(* CODESYS project Estação 7 - Storage (2022).project

Project tree, tasks and I/O mapping:
  Device : CPX-CEC-C1-V3, Festo AG & Co. KG, order no. 3473128, version 3.5.7.37
      unmapped channels: Rotary switch
    application Application
      libraries: Standard, * (System)
      task MainTask (cyclic, interval t#20ms, priority 20) calls PLC_PRG
      program PLC_PRG [ST]
      global variables GVL
      visualisation Visualization_1
      program entrada_pecas [ST]
      program pisca_pisca [ST]
      program home [ST]
      program processo [ST]
      program saida_pecas [ST]
      program atualizar_valores [ST]
      program teste_comunicacao [ST]
    PLC_Diagnosis : PLC-Diagnosis, Festo AG & Co. KG, version 3.5.4.1
    CPX_System : CPX_System, Festo AG & Co. KG, order no. 3473128, version 1.258
      CEC_C1_V3 : CEC-C1-V3, Festo AG & Co. KG, order no. 3473128, version 1.258
          settings:  = 0;  = 232080133852672;  = 1174579392;  = 65535;  = 16885952;  = 13959208;  = 1f5d13d3;  = 5
      _8DI_8DO : 8DI/8DO, Festo AG & Co. KG, order no. 526257, version 1.258
          settings:  = 0;  = 1;  = 1;  = 1;  = 1;  = 0;  = 1;  = 1;  = 0;  = 0;  = 0;  = 0;  = 0;  = 0;  = 0;  = 0;  = 0;  = 0;  = 0;  = 0;  = 0;  = 0;  = 0;  = 0;  = 0;  = 0;  = 0;  = 0;  = 0;  = 0;  = 0;  = 0;  = 0;  = 0;  = 0;  = 0;  = 0;  = 0;  = 0;  = 0;
             = 0;  = 0;  = 0;  = 0;  = 0;  = 0;  = 0;  = 0;  = 0;  = 0;  = 0;  = 0;  = 0;  = 0;  = 0;  = 0;  = 0;  = 0;  = 0;  = 0;  = 0;  = 0;  = 0;  = 0;  = 0;  = 0;  = 0;  = 0;  = 0;  = 0;  = 0;  = 0;  = 0;  = 0;  = 0;  = 0;  = 0;  = 0;  = 0;  = 0;
             = 576751027668385792;  = 'PI%i.0.0.1=1';  = 'PI%i.0.1.1=1';  = 'PI%i.0.2.1=1';  = 'PI%i.1.0.1=1';  = 'PI%i.1.1.1=0';  = 'PI%i.1.4.2=1';  = 'PI%i.1.6.2=1';  = 'PI%i.6.0.1=0';  = 'PI%i.6.1.1=0';  = 'PI%i.6.2.1=0';  = 'PI%i.6.3.1=0';  = 'PI%i.6.4.1=0';  = 'PI%i.6.5.1=0';  = 'PI%i.6.6.1=0';  = 'PI%i.6.7.1=0';  = dd30774a;  = 6
          unmapped channels: Input 0, Output 0
      _8DI_8DO_1 : 8DI/8DO, Festo AG & Co. KG, order no. 526257, version 1.258
          settings:  = 0;  = 1;  = 1;  = 1;  = 1;  = 0;  = 1;  = 1;  = 0;  = 0;  = 0;  = 0;  = 0;  = 0;  = 0;  = 0;  = 0;  = 0;  = 0;  = 0;  = 0;  = 0;  = 0;  = 0;  = 0;  = 0;  = 0;  = 0;  = 0;  = 0;  = 0;  = 0;  = 0;  = 0;  = 0;  = 0;  = 0;  = 0;  = 0;  = 0;
             = 0;  = 0;  = 0;  = 0;  = 0;  = 0;  = 0;  = 0;  = 0;  = 0;  = 0;  = 0;  = 0;  = 0;  = 0;  = 0;  = 0;  = 0;  = 0;  = 0;  = 0;  = 0;  = 0;  = 0;  = 0;  = 0;  = 0;  = 0;  = 0;  = 0;  = 0;  = 0;  = 0;  = 0;  = 0;  = 0;  = 0;  = 0;  = 0;  = 0;
             = 576751027668385792;  = 'PI%i.0.0.1=1';  = 'PI%i.0.1.1=1';  = 'PI%i.0.2.1=1';  = 'PI%i.1.0.1=1';  = 'PI%i.1.1.1=0';  = 'PI%i.1.4.2=1';  = 'PI%i.1.6.2=1';  = 'PI%i.6.0.1=0';  = 'PI%i.6.1.1=0';  = 'PI%i.6.2.1=0';  = 'PI%i.6.3.1=0';  = 'PI%i.6.4.1=0';  = 'PI%i.6.5.1=0';  = 'PI%i.6.6.1=0';  = 'PI%i.6.7.1=0';  = dd39f1d3;  = 6
          unmapped channels: Input 0, Output 0
    Ethernet : Ethernet, 3S - Smart Software Solutions GmbH, version 3.5.10.0
      ModbusTCP_Slave_Device : ModbusTCP Slave Device, 3S - Smart Software Solutions GmbH, version 3.5.10.0
          unmapped channels: Inputs, Outputs
  visualisation Visualization
  text list GlobalTextList
*)

// Device/Application/GVL
{attribute 'qualified_only'}
VAR_GLOBAL
//Entradas
//Sensores
	E_home 	AT %IX1.0 :BOOL; //
	E_error 	 	AT %IX1.1 :BOOL; //
	E_processo	AT %IX1.2 :BOOL; //
	Armazenagem_completada			AT %IX1.3 :BOOL;
	E_provesso 		AT %IX1.4  :BOOL; //
	S_cor 			AT %IX1.5  :BOOL; //Sensor para verificar se a peça é preta
	S_indutivo  	AT %IX1.6  :BOOL; //Sensor indutivo
	//S_indutivodadw 	AT %IX1.7  :BOOL; //Sensor indutivo
//IHM
	Start_btn 		AT	%IX2.0	:BOOL;  //Botão de start
	Stop_btn 		AT	%IX2.1	:BOOL;	//Botão de stop (NF)
	Chave 			AT	%IX2.2	:BOOL;	//Chave auto/manual
	Reset_btn 		AT	%IX2.3	:BOOL;	//Botão de reset
	I4_IHM			AT	%IX2.4	:BOOL;	//Bit de saída 4 da IHM
	I5_IHM			AT	%IX2.5	:BOOL;	//Bit de saída 5 da IHM
	S_Entrada 			AT	%IX2.6	:BOOL;	//Bit de saída 6 da IHM
	I7_IHM			AT	%IX2.7	:BOOL;	//Bit de saída 7 da IHM

	
//Saídas

	//Sinais para o CECC 			
	Fazer_home 	AT	%QX0.0	:BOOL;	//
	Reset_erro 	AT	%QX0.1	:BOOL;	//
	Modo_E_S 	AT	%QX0.2	:BOOL;	//
	B1		 	AT	%QX0.3	:BOOL;	
	B2 			AT	%QX0.4	:BOOL;	//
	B3		 	AT	%QX0.5	:BOOL;	
	gatilho		AT	%QX0.6	:BOOL;	
	Configuracao AT	%QX0.7	:BOOL;	

//IHM				
	Start_LED		AT	%QX1.0	:BOOL;	//LED do botão de start
	Reset_LED 		AT	%QX1.1	:BOOL;	//LED do botão de reset
	Q1_LED 			AT	%QX1.2	:BOOL;	//LED sinalizador Q1
	Q2_LED			AT	%QX1.3	:BOOL;	//LED sinalizador Q2
	E_Saindo		AT	%QX1.5	:BOOL;	//Saída Q4 IHM //Esteira entrando
	E_Entrando		AT	%QX1.4	:BOOL;	//Saída Q5 IHM //Esteira saindo
	Q6_IHM			AT	%QX1.6	:BOOL;	//Saída Q6 IHM
	Q7_IHM 			AT	%QX1.7	:BOOL;	//Saída Q7 IHM
	
	
	flag_btn_visu :BOOL;
	btn_armazena :  BOOL;
	
	B1_Modbus : BOOL;
	B2_Modbus : BOOL;
	B3_Modbus : BOOL;
	
	home: BOOL := FALSE; //Trigger para que a estação reset os erros e faça home
	ligar_pisca: BOOL := FALSE; //Flag para ligar e desligar o pisca pisca
	iniciar_processo: BOOL := FALSE; //Inicia a função de processo, onde pega ou retira a peça de acordo com a flag definir_sentido. Se essa flag estiver setada, é saída. 
	retirar_peca: BOOL := FALSE; //Flag para iniciar processo de retirada da peça (ligar a esteira para retirar a peça da estação 7 e jogar para a 6).
	definir_sentido:	BOOL := FALSE; //Flag para definir se a peça vai entrar ou saír.
	flag_primeira_entrada : BOOL := FALSE; //Flag para ajudar a gerenciar o sinal da saída Q7 da IHM
	estacao_iniciada : BOOL; //Falg para sinalizar que a estação está iniciada 
	estacao_parada: BOOL; //Flag para sinalizar que a estação está parada
	//MODBUS bits
	//Entradas
	Mod_I_0_0 		AT %IX4.0 : BOOL;//start 
	Mod_I_0_1	 	AT %IX4.1 : BOOL;//stop
	Mod_I_0_2 		AT %IX4.2 : BOOL;//reset
	Mod_I_0_3 		AT %IX4.3 : BOOL;//Modo entrada 
	Mod_I_0_4 		AT %IX4.4 : BOOL;//Modo saída 
	Mod_I_0_5 		AT %IX4.5 : BOOL;//Teste resposta da estação - IN 
	Mod_I_0_6 		AT %IX4.6 : BOOL;//B1
	Mod_I_0_7 		AT %IX4.7 : BOOL;//B2		

	Mod_I_1_0 		AT %IX5.0 : BOOL;//B3
	Mod_I_1_1	 	AT %IX5.1 : BOOL;//Iniciar processo
	Mod_I_1_2 		AT %IX5.2 : BOOL;//Confirmação de leitura das cores pela central
	Mod_I_1_3 		AT %IX5.3 : BOOL;
	Mod_I_1_4 		AT %IX5.4 : BOOL;
	Mod_I_1_5 		AT %IX5.5 : BOOL;
	Mod_I_1_6 		AT %IX5.6 : BOOL;
	Mod_I_1_7 		AT %IX5.7 : BOOL;
	
	//Saídas
	Mod_Q_0_0 		AT %QX2.0 : BOOL;//Estação iniciada 	
	Mod_Q_0_1	 	AT %QX2.1 : BOOL;// Estação parada 
	Mod_Q_0_2 		AT %QX2.2 : BOOL;//Estação em processo
	Mod_Q_0_3 		AT %QX2.3 : BOOL;// Estação em modo entrada 
	Mod_Q_0_4 		AT %QX2.4 : BOOL;// Estação em modo saída 
	Mod_Q_0_5 		AT %QX2.5 : BOOL;// Teste resposta da estação - OUT
	Mod_Q_0_6 		AT %QX2.6 : BOOL;//B1 - bit 0 da cor
	Mod_Q_0_7 		AT %QX2.7 : BOOL;//B2 - bit 1 da cor
	
	Mod_Q_1_0 		AT %QX3.0 : BOOL;//B3 - bit 2 da cor
	Mod_Q_1_1 		AT %QX3.1 : BOOL;//Sensor de entrada da estação
	Mod_Q_1_2 		AT %QX3.2 : BOOL;//Cor disponível para leitura
	Mod_Q_1_3 		AT %QX3.3 : BOOL; 
	Mod_Q_1_4 		AT %QX3.4 : BOOL; 
	Mod_Q_1_5	 	AT %QX3.5 : BOOL; 
	Mod_Q_1_6 		AT %QX3.6 : BOOL; 
	Mod_Q_1_7 		AT %QX3.7 : BOOL; 
	
	Mod_Q_2_0 		AT %QX4.0 : BOOL;
	Mod_Q_2_1 		AT %QX4.1 : BOOL;
	Mod_Q_2_2 		AT %QX4.2 : BOOL;
	Mod_Q_2_3 		AT %QX4.3 : BOOL; 
	Mod_Q_2_4 		AT %QX4.4 : BOOL;
	Mod_Q_2_5	 	AT %QX4.5 : BOOL;
	Mod_Q_2_6 		AT %QX4.6 : BOOL; 
	Mod_Q_2_7 		AT %QX4.7 : BOOL; 
	
	Mod_Q_3_0 		AT %QX5.0 : BOOL; //Teste de comunicação - resposta - BIT 24
	Mod_Q_3_1 		AT %QX5.1 : BOOL; 
	Mod_Q_3_2 		AT %QX5.2 : BOOL;
	Mod_Q_3_3 		AT %QX5.3 : BOOL; 
	Mod_Q_3_4 		AT %QX5.4 : BOOL; 
	Mod_Q_3_5	 	AT %QX5.5 : BOOL; 
	Mod_Q_3_6 		AT %QX5.6 : BOOL; 
	Mod_Q_3_7 		AT %QX5.7 : BOOL;
	
END_VAR

// Device/Application/PLC_PRG
PROGRAM PLC_PRG
VAR

	
	
	
END_VAR

atualizar_valores(); //Função que atualiza as variáveis e o MODBUS
pisca_pisca(); //Função que permite o pisca pisca rodar
home(); //Função para fazer o HOME da estação
teste_comunicacao(); //Função para teste de comunicação

IF NOT gvl.estacao_parada AND gvl.estacao_iniciada THEN //Caso a estação não esteja parada e esteja iniciada
	entrada_pecas(); //Função de entrada de peças
	processo(); 	 //Função de processo 
	saida_pecas();   //Função de saída de peças
	gvl.Q1_LED := TRUE; //Liga o LED que indica estação iniciada
ELSE
	gvl.E_Entrando := FALSE; //Reseta flag que indica peça entrando
	gvl.E_Saindo := FALSE;	//Reseta a flag que indica peça saindo	
	gvl.ligar_pisca := FALSE; //Reseta flag que inicia o pisca pisca
	gvl.Q1_LED := FALSE;	 //Apaga o LED que inidca que a estação está iniciada
END_IF

gvl.Modo_E_S := gvl.definir_sentido; //Define entrada ou saída

END_PROGRAM

// Device/Application/atualizar_valores
PROGRAM atualizar_valores
VAR
END_VAR

GVL.Mod_Q_0_0 := GVL.estacao_iniciada; 
GVL.Mod_Q_0_1 := GVL.estacao_parada;
//GVL.Mod_Q_0_2 := GVL.E_processo;
gvl.Mod_Q_0_2 := gvl.ligar_pisca;

IF GVL.definir_sentido THEN
	GVL.Mod_Q_0_3 := FALSE;
	GVL.Mod_Q_0_4 := TRUE;
	ELSE
	GVL.Mod_Q_0_3 := TRUE;
	GVL.Mod_Q_0_4 := FALSE;
END_IF


GVL.Mod_Q_0_6 := GVL.B1_Modbus;
GVL.Mod_Q_0_7 := GVL.B2_Modbus;
GVL.Mod_Q_1_0 := GVL.B3_Modbus;


gvl.iniciar_processo := gvl.Mod_I_1_1; //ATUALIZADO

IF GVL.Mod_I_0_3 AND NOT gvl.Mod_I_0_4 THEN //Sentido de entrada de peças //ATUALIZADO
	gvl.definir_sentido := FALSE;
END_IF

IF NOT GVL.Mod_I_0_3 AND  gvl.Mod_I_0_4 THEN //Sentido de saída de peças //ATUALIZADO
	gvl.definir_sentido := TRUE;
	gvl.B1 := GVL.Mod_I_0_6;//ATUALIZADO
	gvl.B2 := GVL.Mod_I_0_7;//ATUALIZADO
	gvl.B3 := GVL.Mod_I_1_0;//ATUALIZADO
END_IF

IF GVL.Reset_btn OR GVL.Mod_I_0_2 THEN  //Reset geral e home da estação //ATUALIZADO
	gvl.home  := TRUE;
	GVL.estacao_parada := false;
END_IF

IF NOT GVL.Stop_btn OR GVL.Mod_I_0_1 THEN 
	GVL.estacao_parada := TRUE;
END_IF

IF GVL.Start_btn OR GVL.Mod_I_0_0 THEN 
	if not gvl.estacao_parada then
		gvl.estacao_iniciada := true;
	END_IF
END_IF

IF gvl.Mod_I_1_2 THEN
	GVL.B1_Modbus := FALSE;
	GVL.B2_Modbus := FALSE;
	GVL.B3_Modbus := FALSE;
	GVL.Mod_Q_1_2 := FALSE;
END_IF

END_PROGRAM

// Device/Application/home
PROGRAM home
VAR
	
	TON_temp_1: TON;
	TON_1: BOOL;
	TON_temp_2: TON;
	TON_2: BOOL;
	
	passo: INT;

END_VAR

TON_temp_1(IN := TON_1, PT:= T#0.4S);
TON_temp_2(IN := TON_2, PT:= T#0.4S);

IF  gvl.home THEN  //Reset geral da estação
	gvl.ligar_pisca := TRUE;
	GVL.Reset_erro := TRUE;	
	TON_1 := TRUE;
	passo := 1;
	gvl.home := FALSE;
	GVL.Fazer_home := TRUE;	
END_IF

IF TON_temp_1.Q  AND (passo = 1) THEN //Home
	passo := 0;
	GVL.Reset_erro := FALSE;
	GVL.Fazer_home := TRUE;	
	TON_1 := FALSE;
	TON_2 := TRUE;
	passo := 2;
END_IF

IF TON_temp_2.Q  AND  (passo = 2) THEN //Finalização da home
	GVL.Fazer_home := FALSE;	
	TON_2 := FALSE;
	passo := 3;
END_IF

IF (passo = 3) AND NOT gvl.E_processo THEN
	passo := 0;
	gvl.ligar_pisca := FALSE;
END_IF

END_PROGRAM

// Device/Application/pisca_pisca
PROGRAM pisca_pisca
VAR
	
	TON_temp_1: TON;
	TON_1: BOOL;
	TON_temp_2: TON;
	TON_2: BOOL;
	
	passo: INT;
END_VAR

TON_temp_1(IN := TON_1, PT:= T#0.2S);
TON_temp_2(IN := TON_2, PT:= T#0.2S);

IF gvl.ligar_pisca AND (passo = 0)  THEN
	TON_1 := TRUE;
	passo := 1;
END_IF

IF NOT gvl.ligar_pisca THEN
	TON_1 := FALSE;
	TON_2 := FALSE;
	GVL.Q2_LED := FALSE;
	passo := 0;
END_IF

IF TON_temp_1.Q THEN
	TON_1 := FALSE;
	TON_2 := TRUE;
	GVL.Q2_LED := TRUE;
END_IF

IF TON_temp_2.Q THEN
	TON_1 := TRUE;
	TON_2 := FALSE;
	GVL.Q2_LED := FALSE;
END_IF

END_PROGRAM

// Device/Application/teste_comunicacao
PROGRAM teste_comunicacao
VAR
	
	TON_temp_1: TON;
	TON_1: BOOL;	

END_VAR

gvl.Mod_Q_0_5 := gvl.Mod_I_0_5;

END_PROGRAM

// Device/Application/entrada_pecas
PROGRAM entrada_pecas
VAR
	PASSOS_LETURA: INT;
	
	TON_temp_1: TON;
	TON_1: BOOL;
	
	TON_temp_2: TON;
	TON_2: BOOL;
	
	TON_temp_esteira: TON;
	TON_esteira: BOOL;
	
	METALICO: BOOL;
	REFLETE: BOOL;
	
	
END_VAR

TON_temp_1(IN := TON_1, PT:= T#0.4S);
TON_temp_2(IN := TON_2, PT:= T#0.4S);
//Timer para a chagada da peça no sensor da esteira (Esse sensor não está ligado ao CPX, então não consigo utilizar o sinal dele)
TON_temp_esteira(IN := TON_esteira, PT:= T#3S);

IF NOT gvl.definir_sentido AND NOT gvl.E_processo AND NOT gvl.flag_primeira_entrada THEN
	gvl.Q7_IHM := TRUE; 
	gvl.flag_primeira_entrada := TRUE;
END_IF

IF gvl.S_Entrada AND (PASSOS_LETURA = 0) AND NOT gvl.definir_sentido THEN
	gvl.ligar_pisca := TRUE;
	gvl.E_Entrando := TRUE;
	PASSOS_LETURA := 1;
	TON_esteira := TRUE;
	gvl.Q7_IHM := FALSE; 
END_IF

IF (PASSOS_LETURA = 1) AND NOT TON_temp_esteira.Q THEN
	IF NOT METALICO THEN
		METALICO := gvl.S_indutivo;
	END_IF
	IF NOT REFLETE THEN
		REFLETE := gvl.S_cor;
	END_IF
	
END_IF

IF (PASSOS_LETURA = 1) AND  TON_temp_esteira.Q THEN
	
	GVL.B1_Modbus := FALSE;
	GVL.B2_Modbus := FALSE;
	GVL.B3_Modbus := FALSE;
	GVL.Mod_Q_1_2 := FALSE;

	PASSOS_LETURA := 0;
	TON_esteira := FALSE;
	gvl.E_Entrando := FALSE;
	IF METALICO THEN 	
		GVL.B1	:= FALSE;
		GVL.B2	:= TRUE;
		GVL.B3  := FALSE;
	END_IF
	IF NOT METALICO AND REFLETE THEN 	
		GVL.B1	:= FALSE;
		GVL.B2	:= FALSE;
		GVL.B3  := FALSE;
	END_IF
	IF NOT METALICO AND NOT REFLETE THEN 	
		GVL.B1	:= TRUE;
		GVL.B2	:= FALSE;
		GVL.B3  := FALSE;
	END_IF
	
	GVL.B1_Modbus := GVL.B1;
	GVL.B2_Modbus := GVL.B2;
	GVL.B3_Modbus := GVL.B3;
	GVL.Mod_Q_1_2 := TRUE;
	
	METALICO := FALSE;
	REFLETE := FALSE;
	
	PASSOS_LETURA := 2;
END_IF

IF (PASSOS_LETURA = 2) AND NOT gvl.E_processo THEN
	PASSOS_LETURA := 0;
	gvl.iniciar_processo := TRUE;
END_IF

END_PROGRAM

// Device/Application/processo
PROGRAM processo
VAR
	
vetor: INT;
	
	TON_temp_1: TON;
	TON_1: BOOL;
	
	TON_temp_2: TON;
	TON_2: BOOL;
	
	PASSOS: INT;

END_VAR

TON_temp_1(IN := TON_1, PT:= T#0.4S);
TON_temp_2(IN := TON_2, PT:= T#0.4S);

IF NOT gvl.E_processo   AND (GVL.btn_armazena  OR (gvl.iniciar_processo)) THEN
	gvl.iniciar_processo := FALSE;
	gvl.ligar_pisca := TRUE;
	gvl.Configuracao := TRUE;
	TON_1 := TRUE;
	PASSOS := 1;
	
END_IF

IF (PASSOS = 1) AND TON_temp_1.Q THEN
	PASSOS := 2;
	TON_1 := FALSE;
	TON_2 := TRUE;
END_IF

IF (PASSOS = 2) AND TON_temp_2.Q THEN
	PASSOS := 3;
	TON_2 := FALSE;
	gvl.gatilho := TRUE;	
	TON_1 := TRUE;
END_IF

IF (PASSOS = 3) AND TON_temp_1.Q THEN
	PASSOS := 4;
	TON_1 := FALSE;
	gvl.gatilho := FALSE;
	TON_2 := TRUE;
END_IF

IF (PASSOS = 4) AND TON_temp_2.Q THEN
	PASSOS := 5;
	TON_2 := FALSE;
	GVL.B1	:= FALSE;
	GVL.B2	:= FALSE;
	GVL.B3  := FALSE;
END_IF

IF (PASSOS = 5) AND NOT gvl.E_processo THEN
	PASSOS := 0;
	gvl.iniciar_processo := FALSE;
	gvl.ligar_pisca := FALSE;
	gvl.flag_primeira_entrada := FALSE;
	IF gvl.Modo_E_S THEN
		gvl.retirar_peca := TRUE;
	END_IF 
	IF NOT gvl.Modo_E_S THEN
		gvl.Q7_IHM := TRUE;
	END_IF
END_IF

END_PROGRAM

// Device/Application/saida_pecas
PROGRAM saida_pecas
VAR

	PASSOS: INT;
	
	TON_temp_esteira: TON;
	TON_esteira: BOOL;
	
	TON_temp_1: TON;
	TON_1: BOOL;	
	
	METALICO: BOOL;
	REFLETE: BOOL;	

END_VAR

TON_temp_1(IN := TON_1, PT:= T#0.8S);
//Timer para a chagada da peça no sensor da esteira (Esse sensor não está ligado ao CPX, então não consigo utilizar o sinal dele)
TON_temp_esteira(IN := TON_esteira, PT:= T#3S);

IF gvl.retirar_peca AND (PASSOS = 0)THEN
	gvl.retirar_peca := FALSE;
	gvl.ligar_pisca := TRUE;
	gvl.E_saindo := TRUE;
	gvl.Q7_IHM := FALSE;
	PASSOS := 1;
END_IF

IF (PASSOS = 1) AND gvl.S_Entrada THEN
	gvl.ligar_pisca := FALSE;
	TON_1 := TRUE;
	gvl.Q7_IHM := TRUE;
	TON_esteira := TRUE;
	PASSOS := 2;
END_IF

IF TON_temp_1.Q THEN
	TON_1 := FALSE;
	gvl.Q7_IHM := FALSE;
END_IF

IF (PASSOS = 2) AND TON_temp_esteira.Q THEN
	TON_esteira := FALSE;
	gvl.E_saindo := FALSE;
	PASSOS := 0;
END_IF

END_PROGRAM

// /Visualization
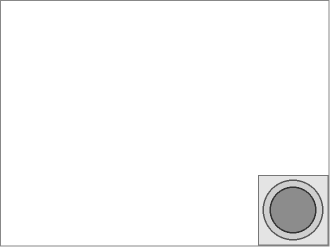
VISUALIZATION Visualization  // 330x247
    PushSwitch (258,175 70x70), variable: GVL.flag_btn_visu, behaviour: TOGGLE, style: Switch-PushSwitch-Gray
END_VISUALIZATION

// Device/Application/Visualization_1
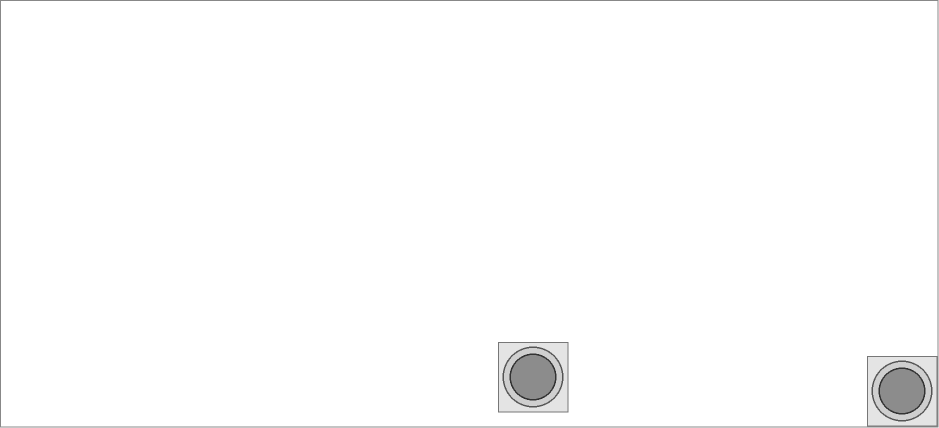
VISUALIZATION Visualization_1  // 939x428
    PushSwitch (498,342 70x70), variable: GVL.flag_btn_visu, behaviour: TAP, style: Switch-PushSwitch-Gray
    PushSwitch (867,356 70x70), variable: GVL.btn_armazena, behaviour: TAP, style: Switch-PushSwitch-Gray
END_VISUALIZATION
